// TIA Portal V18 export
// export: Created 2025-06-15T08:30:00, ExportSetting WithDefaults
DATA_BLOCK "DB5_Filler"   // DB5
{ S7_Optimized_Access := 'FALSE' }
BEGIN
END_DATA_BLOCK

DATA_BLOCK "DB6_Capper"   // DB6
{ S7_Optimized_Access := 'FALSE' }
BEGIN
END_DATA_BLOCK

DATA_BLOCK "DB7_Labeler"   // DB7
{ S7_Optimized_Access := 'FALSE' }
BEGIN
END_DATA_BLOCK

DATA_BLOCK "DB8_Conveyor"   // DB8
{ S7_Optimized_Access := 'FALSE' }
BEGIN
END_DATA_BLOCK

DATA_BLOCK "DB10_Production"   // DB10
{ S7_Optimized_Access := 'FALSE' }
BEGIN
END_DATA_BLOCK

VAR_GLOBAL   // PLC tag table "BottlingLine_IO"
END_VAR
